{attribute 'GeneratedUsingTerminal: EL2732-0000-0016'}
{attribute addProperty BoxType "EL2732-0000-0016"}
{attribute addProperty Id "Channel_1AT %Q*Channel_42CA91F71Channel_2AT %Q*Channel_42CA91F71WcStateAT %I*WcState_0B2B16F91InfoDataAT %I*InfoData_6F19DB2B2"}
{attribute addProperty CRC "2954971456"}
{attribute addProperty Size "5"}
TYPE EL2732_B0214940 EXTENDS EtcSlaveTerminalBase_947E5A46 :
STRUCT
	{attribute addProperty Name "Channel_1"}
	Channel_1 : Channel_42CA91F7;
	{attribute addProperty Name "Channel_2"}
	Channel_2 : Channel_42CA91F7;
	{attribute addProperty Name "WcState"}
	WcState : WcState_0B2B16F9;
	{attribute addProperty Name "InfoData"}
	InfoData : InfoData_6F19DB2B;
END_STRUCT
END_TYPE

(* stored: Version 1.2.0.0, ProductVersion 3.1.4024.9
   DUT EL2732_B0214940: Id {e448858f-12d7-4baa-ad8a-80b7f678d195} *)
